FUNCTION_BLOCK PROD_MAN
  {SET_ATTRIBUTE(OpcUa, SERVICE)}
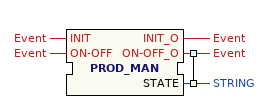
  EVENT_INPUT
    INIT;
    ON-OFF;
  END_EVENT
  EVENT_OUTPUT
    INIT_O;
    ON-OFF_O WITH STATE;
  END_EVENT
  VAR_OUTPUT
    STATE : STRING;
  END_VAR
END_FUNCTION_BLOCK
